TYPE ST_LEDSystem :
STRUCT
	stLED_r: ST_LED := (color:='RED');
	stLED_o: ST_LED := (color:='ORANGE');
	stLED_g: ST_LED := (color:='GREEN');
	arrLog: ARRAY [0..20] OF ST_Log;
	stRequest_r: ST_Request := ();
	stRequest_o: ST_Request := ();
	stRequest_g: ST_Request := ();
END_STRUCT
END_TYPE

(* stored: Version 1.1.0.1, ProductVersion 3.1.4022.12
   DUT ST_LEDSystem: Id {7c3a5aa1-adab-48e5-b322-9f65d05a9cb5} *)
